ABB RAPID module: Module1.mod

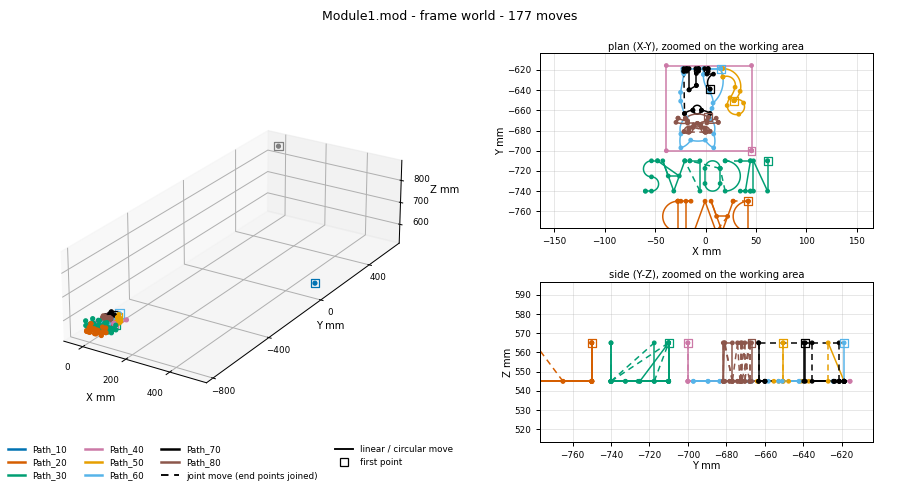
[picture p0: tool path of Module1.mod in frame world, 177 of 177 moves have a stored position in this frame; points joined in program order, loops and branches not executed]
MODULE Module1
    CONST robtarget Target_home:=[[-424.990093119,-612,35.499184826],[0,0.996194698,0,0.087155743],[0,0,0,0],[9E+09,9E+09,9E+09,9E+09,9E+09,9E+09]];
    CONST robtarget D1A:=[[68.121,138,20],[0,-0.707106781,0.707106781,0],[0,0,0,0],[9E+09,9E+09,9E+09,9E+09,9E+09,9E+09]];
    CONST robtarget D11:=[[68.121,138,0],[0,-0.707106781,0.707106781,0],[0,0,0,0],[9E+09,9E+09,9E+09,9E+09,9E+09,9E+09]];
    CONST robtarget D12:=[[68.121,168,0],[0,-0.707106781,0.707106781,0],[0,0,0,0],[9E+09,9E+09,9E+09,9E+09,9E+09,9E+09]];
    CONST robtarget D13:=[[83.121,153,0],[0,-0.707106781,0.707106781,0],[0,0,0,0],[9E+09,9E+09,9E+09,9E+09,9E+09,9E+09]];
    CONST robtarget A1A:=[[83.121,138,20],[0,-0.707106781,0.707106781,0],[0,0,0,0],[9E+09,9E+09,9E+09,9E+09,9E+09,9E+09]];
    CONST robtarget A11:=[[83.121,138,0],[0,-0.707106781,0.707106781,0],[0,0,0,0],[9E+09,9E+09,9E+09,9E+09,9E+09,9E+09]];
    CONST robtarget A12:=[[94.04,168,0],[0,-0.707106781,0.707106781,0],[0,0,0,0],[9E+09,9E+09,9E+09,9E+09,9E+09,9E+09]];
    CONST robtarget A13:=[[104.96,138,0],[0,-0.707106781,0.707106781,0],[0,0,0,0],[9E+09,9E+09,9E+09,9E+09,9E+09,9E+09]];
    CONST robtarget A14:=[[99.5,153,0],[0,-0.707106781,0.707106781,0],[0,0,0,0],[9E+09,9E+09,9E+09,9E+09,9E+09,9E+09]];
    CONST robtarget A15:=[[88.581,153,0],[0,-0.707106781,0.707106781,0],[0,0,0,0],[9E+09,9E+09,9E+09,9E+09,9E+09,9E+09]];
    CONST robtarget VA:=[[100.04,168,20],[0,-0.707106781,0.707106781,0],[0,0,0,0],[9E+09,9E+09,9E+09,9E+09,9E+09,9E+09]];
    CONST robtarget V1:=[[100.04,168,0],[0,-0.707106781,0.707106781,0],[0,0,0,0],[9E+09,9E+09,9E+09,9E+09,9E+09,9E+09]];
    CONST robtarget V2:=[[110.96,138,0],[0,-0.707106781,0.707106781,0],[0,0,0,0],[9E+09,9E+09,9E+09,9E+09,9E+09,9E+09]];
    CONST robtarget V3:=[[121.879,168,0],[0,-0.707106781,0.707106781,0],[0,0,0,0],[9E+09,9E+09,9E+09,9E+09,9E+09,9E+09]];
    CONST robtarget I1A:=[[124.879,168,20],[0,-0.707106781,0.707106781,0],[0,0,0,0],[9E+09,9E+09,9E+09,9E+09,9E+09,9E+09]];
    CONST robtarget I11:=[[124.879,168,0],[0,-0.707106781,0.707106781,0],[0,0,0,0],[9E+09,9E+09,9E+09,9E+09,9E+09,9E+09]];
    CONST robtarget I12:=[[134.879,168,0],[0,-0.707106781,0.707106781,0],[0,0,0,0],[9E+09,9E+09,9E+09,9E+09,9E+09,9E+09]];
    CONST robtarget I13:=[[129.879,168,0],[0,-0.707106781,0.707106781,0],[0,0,0,0],[9E+09,9E+09,9E+09,9E+09,9E+09,9E+09]];
    CONST robtarget I14:=[[129.879,138,0],[0,-0.707106781,0.707106781,0],[0,0,0,0],[9E+09,9E+09,9E+09,9E+09,9E+09,9E+09]];
    CONST robtarget I15:=[[124.879,138,0],[0,-0.707106781,0.707106781,0],[0,0,0,0],[9E+09,9E+09,9E+09,9E+09,9E+09,9E+09]];
    CONST robtarget I16:=[[134.879,138,0],[0,-0.707106781,0.707106781,0],[0,0,0,0],[9E+09,9E+09,9E+09,9E+09,9E+09,9E+09]];
    CONST robtarget D2A:=[[137.879,138,20],[0,-0.707106781,0.707106781,0],[0,0,0,0],[9E+09,9E+09,9E+09,9E+09,9E+09,9E+09]];
    CONST robtarget D21:=[[137.879,138,0],[0,-0.707106781,0.707106781,0],[0,0,0,0],[9E+09,9E+09,9E+09,9E+09,9E+09,9E+09]];
    CONST robtarget D22:=[[137.879,168,0],[0,-0.707106781,0.707106781,0],[0,0,0,0],[9E+09,9E+09,9E+09,9E+09,9E+09,9E+09]];
    CONST robtarget D23:=[[152.879,153,0],[0,-0.707106781,0.707106781,0],[0,0,0,0],[9E+09,9E+09,9E+09,9E+09,9E+09,9E+09]];
    PERS tooldata PM:=[TRUE,[[71.138,0,74.787],[0.819152044,0,0.573576436,0]],[1,[0,0,1],[1,0,0,0],0,0,0]];
    TASK PERS wobjdata Pastel:=[FALSE,TRUE,"",[[0,0,0],[1,0,0,0]],[[110.5,-612,545],[0,0,0,1]]];
    CONST robtarget SA:=[[158.029,98,20],[0,-0.707106781,0.707106781,0],[0,0,0,0],[9E+09,9E+09,9E+09,9E+09,9E+09,9E+09]];
    CONST robtarget CA:=[[91.029,98,20],[0,-0.707106781,0.707106781,0],[0,0,0,0],[9E+09,9E+09,9E+09,9E+09,9E+09,9E+09]];
    CONST robtarget C1:=[[91.029,98,0],[0,-0.707106781,0.707106781,0],[0,0,0,0],[9E+09,9E+09,9E+09,9E+09,9E+09,9E+09]];
    CONST robtarget C2:=[[76.029,113,0],[0,-0.707106781,0.707106781,0],[0,0,0,0],[9E+09,9E+09,9E+09,9E+09,9E+09,9E+09]];
    CONST robtarget C3:=[[91.029,128,0],[0,-0.707106781,0.707106781,0],[0,0,0,0],[9E+09,9E+09,9E+09,9E+09,9E+09,9E+09]];
    CONST robtarget OA:=[[96.029,105.5,20],[0,-0.707106781,0.707106781,0],[0,0,0,0],[9E+09,9E+09,9E+09,9E+09,9E+09,9E+09]];
    CONST robtarget O1:=[[96.029,105.5,0],[0,-0.707106781,0.707106781,0],[0,0,0,0],[9E+09,9E+09,9E+09,9E+09,9E+09,9E+09]];
    CONST robtarget O2:=[[96.029,120.5,0],[0,-0.707106781,0.707106781,0],[0,0,0,0],[9E+09,9E+09,9E+09,9E+09,9E+09,9E+09]];
    CONST robtarget O3:=[[103.529,128,0],[0,-0.707106781,0.707106781,0],[0,0,0,0],[9E+09,9E+09,9E+09,9E+09,9E+09,9E+09]];
    CONST robtarget O4:=[[111.029,120.5,0],[0,-0.707106781,0.707106781,0],[0,0,0,0],[9E+09,9E+09,9E+09,9E+09,9E+09,9E+09]];
    CONST robtarget O5:=[[111.029,105.5,0],[0,-0.707106781,0.707106781,0],[0,0,0,0],[9E+09,9E+09,9E+09,9E+09,9E+09,9E+09]];
    CONST robtarget O6:=[[103.529,98,0],[0,-0.707106781,0.707106781,0],[0,0,0,0],[9E+09,9E+09,9E+09,9E+09,9E+09,9E+09]];
    CONST robtarget LA:=[[126.029,98,20],[0,-0.707106781,0.707106781,0],[0,0,0,0],[9E+09,9E+09,9E+09,9E+09,9E+09,9E+09]];
    CONST robtarget L1:=[[126.029,98,0],[0,-0.707106781,0.707106781,0],[0,0,0,0],[9E+09,9E+09,9E+09,9E+09,9E+09,9E+09]];
    CONST robtarget L2:=[[116.029,98,0],[0,-0.707106781,0.707106781,0],[0,0,0,0],[9E+09,9E+09,9E+09,9E+09,9E+09,9E+09]];
    CONST robtarget L3:=[[116.029,128,0],[0,-0.707106781,0.707106781,0],[0,0,0,0],[9E+09,9E+09,9E+09,9E+09,9E+09,9E+09]];
    CONST robtarget A2A:=[[131.029,98,20],[0,-0.707106781,0.707106781,0],[0,0,0,0],[9E+09,9E+09,9E+09,9E+09,9E+09,9E+09]];
    CONST robtarget A21:=[[131.029,98,0],[0,-0.707106781,0.707106781,0],[0,0,0,0],[9E+09,9E+09,9E+09,9E+09,9E+09,9E+09]];
    CONST robtarget A22:=[[141.948,128,0],[0,-0.707106781,0.707106781,0],[0,0,0,0],[9E+09,9E+09,9E+09,9E+09,9E+09,9E+09]];
    CONST robtarget A23:=[[152.867,98,0],[0,-0.707106781,0.707106781,0],[0,0,0,0],[9E+09,9E+09,9E+09,9E+09,9E+09,9E+09]];
    CONST robtarget A24:=[[147.408,113,0],[0,-0.707106781,0.707106781,0],[0,0,0,0],[9E+09,9E+09,9E+09,9E+09,9E+09,9E+09]];
    CONST robtarget A25:=[[136.489,113,0],[0,-0.707106781,0.707106781,0],[0,0,0,0],[9E+09,9E+09,9E+09,9E+09,9E+09,9E+09]];
    CONST robtarget S1:=[[158.029,98,0],[0,-0.707106781,0.707106781,0],[0,0,0,0],[9E+09,9E+09,9E+09,9E+09,9E+09,9E+09]];
    CONST robtarget S2:=[[164.029,98,0],[0,-0.707106781,0.707106781,0],[0,0,0,0],[9E+09,9E+09,9E+09,9E+09,9E+09,9E+09]];
    CONST robtarget S3:=[[171.971,105.942,0],[0,-0.707106781,0.707106781,0],[0,0,0,0],[9E+09,9E+09,9E+09,9E+09,9E+09,9E+09]];
    CONST robtarget S4:=[[164.029,113.883,0],[0,-0.707106781,0.707106781,0],[0,0,0,0],[9E+09,9E+09,9E+09,9E+09,9E+09,9E+09]];
    CONST robtarget S5:=[[156.971,120.942,0],[0,-0.707106781,0.707106781,0],[0,0,0,0],[9E+09,9E+09,9E+09,9E+09,9E+09,9E+09]];
    CONST robtarget S6:=[[164.029,128,0],[0,-0.707106781,0.707106781,0],[0,0,0,0],[9E+09,9E+09,9E+09,9E+09,9E+09,9E+09]];
    CONST robtarget S7:=[[170.029,128,0],[0,-0.707106781,0.707106781,0],[0,0,0,0],[9E+09,9E+09,9E+09,9E+09,9E+09,9E+09]];
    CONST robtarget SF:=[[170.029,128,20],[0,-0.707106781,0.707106781,0],[0,0,0,0],[9E+09,9E+09,9E+09,9E+09,9E+09,9E+09]];
    CONST robtarget NA:=[[49.029,98,20],[0,-0.707106781,0.707106781,0],[0,0,0,0],[9E+09,9E+09,9E+09,9E+09,9E+09,9E+09]];
    CONST robtarget N4:=[[63.029,128,0],[0,-0.707106781,0.707106781,0],[0,0,0,0],[9E+09,9E+09,9E+09,9E+09,9E+09,9E+09]];
    CONST robtarget N3:=[[63.029,98,0],[0,-0.707106781,0.707106781,0],[0,0,0,0],[9E+09,9E+09,9E+09,9E+09,9E+09,9E+09]];
    CONST robtarget N2:=[[49.029,128,0],[0,-0.707106781,0.707106781,0],[0,0,0,0],[9E+09,9E+09,9E+09,9E+09,9E+09,9E+09]];
    CONST robtarget N1:=[[49.029,98,0],[0,-0.707106781,0.707106781,0],[0,0,0,0],[9E+09,9E+09,9E+09,9E+09,9E+09,9E+09]];
    CONST robtarget I26:=[[76.029,98,0],[0,-0.707106781,0.707106781,0],[0,0,0,0],[9E+09,9E+09,9E+09,9E+09,9E+09,9E+09]];
    CONST robtarget I25:=[[66.029,98,0],[0,-0.707106781,0.707106781,0],[0,0,0,0],[9E+09,9E+09,9E+09,9E+09,9E+09,9E+09]];
    CONST robtarget I24:=[[71.029,98,0],[0,-0.707106781,0.707106781,0],[0,0,0,0],[9E+09,9E+09,9E+09,9E+09,9E+09,9E+09]];
    CONST robtarget I23:=[[71.029,128,0],[0,-0.707106781,0.707106781,0],[0,0,0,0],[9E+09,9E+09,9E+09,9E+09,9E+09,9E+09]];
    CONST robtarget I22:=[[76.029,128,0],[0,-0.707106781,0.707106781,0],[0,0,0,0],[9E+09,9E+09,9E+09,9E+09,9E+09,9E+09]];
    CONST robtarget I21:=[[66.029,128,0],[0,-0.707106781,0.707106781,0],[0,0,0,0],[9E+09,9E+09,9E+09,9E+09,9E+09,9E+09]];
    CONST robtarget I2A:=[[66.029,128,20],[0,-0.707106781,0.707106781,0],[0,0,0,0],[9E+09,9E+09,9E+09,9E+09,9E+09,9E+09]];
    CONST robtarget CUAA:=[[64.919,88,20],[0,-0.707106781,0.707106781,0],[0,0,0,0],[9E+09,9E+09,9E+09,9E+09,9E+09,9E+09]];
    CONST robtarget E1:=[[64.919,88,0],[0,-0.707106781,0.707106781,0],[0,0,0,0],[9E+09,9E+09,9E+09,9E+09,9E+09,9E+09]];
    CONST robtarget E2:=[[149.319,88,0],[0,-0.707106781,0.707106781,0],[0,0,0,0],[9E+09,9E+09,9E+09,9E+09,9E+09,9E+09]];
    CONST robtarget E3:=[[149.319,3.6,0],[0,-0.707106781,0.707106781,0],[0,0,0,0],[9E+09,9E+09,9E+09,9E+09,9E+09,9E+09]];
    CONST robtarget E4:=[[64.919,3.6,0],[0,-0.707106781,0.707106781,0],[0,0,0,0],[9E+09,9E+09,9E+09,9E+09,9E+09,9E+09]];
    CONST robtarget P11:=[[82.21,38.425,20],[0,-0.707106781,0.707106781,0],[0,0,0,0],[9E+09,9E+09,9E+09,9E+09,9E+09,9E+09]];
    CONST robtarget P12:=[[82.21,38.425,0],[0,-0.707106781,0.707106781,0],[0,0,0,0],[9E+09,9E+09,9E+09,9E+09,9E+09,9E+09]];
    CONST robtarget P13:=[[76.99,37.487,0],[0,-0.707106781,0.707106781,0],[0,0,0,0],[9E+09,9E+09,9E+09,9E+09,9E+09,9E+09]];
    CONST robtarget P14:=[[72.798,40.737,0],[0,-0.707106781,0.707106781,0],[0,0,0,0],[9E+09,9E+09,9E+09,9E+09,9E+09,9E+09]];
    CONST robtarget P15:=[[72.498,47.446,0],[0,-0.707106781,0.707106781,0],[0,0,0,0],[9E+09,9E+09,9E+09,9E+09,9E+09,9E+09]];
    CONST robtarget P16:=[[77.549,51.872,0],[0,-0.707106781,0.707106781,0],[0,0,0,0],[9E+09,9E+09,9E+09,9E+09,9E+09,9E+09]];
    CONST robtarget P17:=[[85.419,50.387,0],[0,-0.707106781,0.707106781,0],[0,0,0,0],[9E+09,9E+09,9E+09,9E+09,9E+09,9E+09]];
    CONST robtarget P18:=[[89.032,43.239,0],[0,-0.707106781,0.707106781,0],[0,0,0,0],[9E+09,9E+09,9E+09,9E+09,9E+09,9E+09]];
    CONST robtarget P19:=[[88.217,39.173,0],[0,-0.707106781,0.707106781,0],[0,0,0,0],[9E+09,9E+09,9E+09,9E+09,9E+09,9E+09]];
    CONST robtarget P110:=[[86.183,35.559,0],[0,-0.707106781,0.707106781,0],[0,0,0,0],[9E+09,9E+09,9E+09,9E+09,9E+09,9E+09]];
    CONST robtarget P111:=[[83.19,30.571,0],[0,-0.707106781,0.707106781,0],[0,0,0,0],[9E+09,9E+09,9E+09,9E+09,9E+09,9E+09]];
    CONST robtarget P112:=[[81.2,25.106,0],[0,-0.707106781,0.707106781,0],[0,0,0,0],[9E+09,9E+09,9E+09,9E+09,9E+09,9E+09]];
    CONST robtarget P113:=[[84.037,16.23,0],[0,-0.707106781,0.707106781,0],[0,0,0,0],[9E+09,9E+09,9E+09,9E+09,9E+09,9E+09]];
    CONST robtarget P114:=[[93.269,14.968,0],[0,-0.707106781,0.707106781,0],[0,0,0,0],[9E+09,9E+09,9E+09,9E+09,9E+09,9E+09]];
    CONST robtarget P115:=[[93.269,14.968,20],[0,-0.707106781,0.707106781,0],[0,0,0,0],[9E+09,9E+09,9E+09,9E+09,9E+09,9E+09]];
    CONST robtarget P116:=[[95.609,6.67,0],[0,-0.707106781,0.707106781,0],[0,0,0,0],[9E+09,9E+09,9E+09,9E+09,9E+09,9E+09]];
    CONST robtarget P117:=[[93.269,6.67,0],[0,-0.707106781,0.707106781,0],[0,0,0,0],[9E+09,9E+09,9E+09,9E+09,9E+09,9E+09]];
    CONST robtarget P118:=[[79.171,13.675,0],[0,-0.707106781,0.707106781,0],[0,0,0,0],[9E+09,9E+09,9E+09,9E+09,9E+09,9E+09]];
    CONST robtarget P119:=[[76.238,29.142,0],[0,-0.707106781,0.707106781,0],[0,0,0,0],[9E+09,9E+09,9E+09,9E+09,9E+09,9E+09]];
    CONST robtarget P120:=[[78.528,34.232,0],[0,-0.707106781,0.707106781,0],[0,0,0,0],[9E+09,9E+09,9E+09,9E+09,9E+09,9E+09]];
    CONST robtarget P232:=[[103.027,40.737,0],[0,-0.707106781,0.707106781,0],[0,0,0,0],[9E+09,9E+09,9E+09,9E+09,9E+09,9E+09]];
    CONST robtarget P210:=[[135.23,62.86,0],[0,-0.707106781,0.707106781,0],[0,0,0,0],[9E+09,9E+09,9E+09,9E+09,9E+09,9E+09]];
    CONST robtarget P211:=[[134.911,71.377,0],[0,-0.707106781,0.707106781,0],[0,0,0,0],[9E+09,9E+09,9E+09,9E+09,9E+09,9E+09]];
    CONST robtarget P212:=[[135.861,78.258,0],[0,-0.707106781,0.707106781,0],[0,0,0,0],[9E+09,9E+09,9E+09,9E+09,9E+09,9E+09]];
    CONST robtarget P213:=[[134.911,85.138,0],[0,-0.707106781,0.707106781,0],[0,0,0,0],[9E+09,9E+09,9E+09,9E+09,9E+09,9E+09]];
    CONST robtarget P214:=[[129.352,82.199,0],[0,-0.707106781,0.707106781,0],[0,0,0,0],[9E+09,9E+09,9E+09,9E+09,9E+09,9E+09]];
    CONST robtarget P215:=[[125.181,77.493,0],[0,-0.707106781,0.707106781,0],[0,0,0,0],[9E+09,9E+09,9E+09,9E+09,9E+09,9E+09]];
    CONST robtarget P216:=[[117.953,78.45,0],[0,-0.707106781,0.707106781,0],[0,0,0,0],[9E+09,9E+09,9E+09,9E+09,9E+09,9E+09]];
    CONST robtarget P217:=[[110.724,77.493,0],[0,-0.707106781,0.707106781,0],[0,0,0,0],[9E+09,9E+09,9E+09,9E+09,9E+09,9E+09]];
    CONST robtarget P218:=[[107.111,81.908,0],[0,-0.707106781,0.707106781,0],[0,0,0,0],[9E+09,9E+09,9E+09,9E+09,9E+09,9E+09]];
    CONST robtarget P219:=[[102.4,85.125,0],[0,-0.707106781,0.707106781,0],[0,0,0,0],[9E+09,9E+09,9E+09,9E+09,9E+09,9E+09]];
    CONST robtarget P220:=[[101.194,78.244,0],[0,-0.707106781,0.707106781,0],[0,0,0,0],[9E+09,9E+09,9E+09,9E+09,9E+09,9E+09]];
    CONST robtarget P221:=[[102.4,71.363,0],[0,-0.707106781,0.707106781,0],[0,0,0,0],[9E+09,9E+09,9E+09,9E+09,9E+09,9E+09]];
    CONST robtarget P222:=[[101.604,63.136,0],[0,-0.707106781,0.707106781,0],[0,0,0,0],[9E+09,9E+09,9E+09,9E+09,9E+09,9E+09]];
    CONST robtarget P223:=[[105.943,56.102,0],[0,-0.707106781,0.707106781,0],[0,0,0,0],[9E+09,9E+09,9E+09,9E+09,9E+09,9E+09]];
    CONST robtarget P224:=[[107.614,54.857,0],[0,-0.707106781,0.707106781,0],[0,0,0,0],[9E+09,9E+09,9E+09,9E+09,9E+09,9E+09]];
    CONST robtarget P225:=[[104.069,46.093,0],[0,-0.707106781,0.707106781,0],[0,0,0,0],[9E+09,9E+09,9E+09,9E+09,9E+09,9E+09]];
    CONST robtarget P226:=[[103.223,37.713,0],[0,-0.707106781,0.707106781,0],[0,0,0,0],[9E+09,9E+09,9E+09,9E+09,9E+09,9E+09]];
    CONST robtarget P227:=[[106.607,30,0],[0,-0.707106781,0.707106781,0],[0,0,0,0],[9E+09,9E+09,9E+09,9E+09,9E+09,9E+09]];
    CONST robtarget P228:=[[111.198,21.776,0],[0,-0.707106781,0.707106781,0],[0,0,0,0],[9E+09,9E+09,9E+09,9E+09,9E+09,9E+09]];
    CONST robtarget P229:=[[112.662,12.472,0],[0,-0.707106781,0.707106781,0],[0,0,0,0],[9E+09,9E+09,9E+09,9E+09,9E+09,9E+09]];
    CONST robtarget P230:=[[112.476,6.67,0],[0,-0.707106781,0.707106781,0],[0,0,0,0],[9E+09,9E+09,9E+09,9E+09,9E+09,9E+09]];
    CONST robtarget P231:=[[93.703,24.926,0],[0,-0.707106781,0.707106781,0],[0,0,0,0],[9E+09,9E+09,9E+09,9E+09,9E+09,9E+09]];
    CONST robtarget P29:=[[129.718,55.201,0],[0,-0.707106781,0.707106781,0],[0,0,0,0],[9E+09,9E+09,9E+09,9E+09,9E+09,9E+09]];
    CONST robtarget P28:=[[132.81,47.291,0],[0,-0.707106781,0.707106781,0],[0,0,0,0],[9E+09,9E+09,9E+09,9E+09,9E+09,9E+09]];
    CONST robtarget P27:=[[135.088,38.885,0],[0,-0.707106781,0.707106781,0],[0,0,0,0],[9E+09,9E+09,9E+09,9E+09,9E+09,9E+09]];
    CONST robtarget P26:=[[135.236,30.178,0],[0,-0.707106781,0.707106781,0],[0,0,0,0],[9E+09,9E+09,9E+09,9E+09,9E+09,9E+09]];
    CONST robtarget P25:=[[131.968,12.02,0],[0,-0.707106781,0.707106781,0],[0,0,0,0],[9E+09,9E+09,9E+09,9E+09,9E+09,9E+09]];
    CONST robtarget P24:=[[134.388,9.719,0],[0,-0.707106781,0.707106781,0],[0,0,0,0],[9E+09,9E+09,9E+09,9E+09,9E+09,9E+09]];
    CONST robtarget P23:=[[133.026,6.67,0],[0,-0.707106781,0.707106781,0],[0,0,0,0],[9E+09,9E+09,9E+09,9E+09,9E+09,9E+09]];
    CONST robtarget P22:=[[95.609,6.67,0],[0,-0.707106781,0.707106781,0],[0,0,0,0],[9E+09,9E+09,9E+09,9E+09,9E+09,9E+09]];
    CONST robtarget P21:=[[95.609,6.67,20],[0,-0.707106781,0.707106781,0],[0,0,0,0],[9E+09,9E+09,9E+09,9E+09,9E+09,9E+09]];
    CONST robtarget P31:=[[106.008,26.905,20],[0,-0.707106781,0.707106781,0],[0,0,0,0],[9E+09,9E+09,9E+09,9E+09,9E+09,9E+09]];
    CONST robtarget P32:=[[106.008,26.905,0],[0,-0.707106781,0.707106781,0],[0,0,0,0],[9E+09,9E+09,9E+09,9E+09,9E+09,9E+09]];
    CONST robtarget P33:=[[108.265,18.63,0],[0,-0.707106781,0.707106781,0],[0,0,0,0],[9E+09,9E+09,9E+09,9E+09,9E+09,9E+09]];
    CONST robtarget P34:=[[102.665,12.134,0],[0,-0.707106781,0.707106781,0],[0,0,0,0],[9E+09,9E+09,9E+09,9E+09,9E+09,9E+09]];
    CONST robtarget P35:=[[109.043,12.02,0],[0,-0.707106781,0.707106781,0],[0,0,0,0],[9E+09,9E+09,9E+09,9E+09,9E+09,9E+09]];
    CONST robtarget P36:=[[111.486,9.9,0],[0,-0.707106781,0.707106781,0],[0,0,0,0],[9E+09,9E+09,9E+09,9E+09,9E+09,9E+09]];
    CONST robtarget P37:=[[111.341,6.67,0],[0,-0.707106781,0.707106781,0],[0,0,0,0],[9E+09,9E+09,9E+09,9E+09,9E+09,9E+09]];
    CONST robtarget P38:=[[107.849,6.67,0],[0,-0.707106781,0.707106781,0],[0,0,0,0],[9E+09,9E+09,9E+09,9E+09,9E+09,9E+09]];
    CONST robtarget P39:=[[107.849,9.239,0],[0,-0.707106781,0.707106781,0],[0,0,0,0],[9E+09,9E+09,9E+09,9E+09,9E+09,9E+09]];
    CONST robtarget P310:=[[117.381,6.67,0],[0,-0.707106781,0.707106781,0],[0,0,0,0],[9E+09,9E+09,9E+09,9E+09,9E+09,9E+09]];
    CONST robtarget P311:=[[117.381,9.136,0],[0,-0.707106781,0.707106781,0],[0,0,0,0],[9E+09,9E+09,9E+09,9E+09,9E+09,9E+09]];
    CONST robtarget P312:=[[120.124,6.67,0],[0,-0.707106781,0.707106781,0],[0,0,0,0],[9E+09,9E+09,9E+09,9E+09,9E+09,9E+09]];
    CONST robtarget P313:=[[121.413,9.237,0],[0,-0.707106781,0.707106781,0],[0,0,0,0],[9E+09,9E+09,9E+09,9E+09,9E+09,9E+09]];
    CONST robtarget P314:=[[119.569,11.44,0],[0,-0.707106781,0.707106781,0],[0,0,0,0],[9E+09,9E+09,9E+09,9E+09,9E+09,9E+09]];
    CONST robtarget P315:=[[119.569,23.339,0],[0,-0.707106781,0.707106781,0],[0,0,0,0],[9E+09,9E+09,9E+09,9E+09,9E+09,9E+09]];
    CONST robtarget P316:=[[119.569,23.339,20],[0,-0.707106781,0.707106781,0],[0,0,0,0],[9E+09,9E+09,9E+09,9E+09,9E+09,9E+09]];
    CONST robtarget P317:=[[126.788,27.654,20],[0,-0.707106781,0.707106781,0],[0,0,0,0],[9E+09,9E+09,9E+09,9E+09,9E+09,9E+09]];
    CONST robtarget P318:=[[126.788,27.654,0],[0,-0.707106781,0.707106781,0],[0,0,0,0],[9E+09,9E+09,9E+09,9E+09,9E+09,9E+09]];
    CONST robtarget P319:=[[126.788,6.67,0],[0,-0.707106781,0.707106781,0],[0,0,0,0],[9E+09,9E+09,9E+09,9E+09,9E+09,9E+09]];
    CONST robtarget P320:=[[129.217,6.67,0],[0,-0.707106781,0.707106781,0],[0,0,0,0],[9E+09,9E+09,9E+09,9E+09,9E+09,9E+09]];
    CONST robtarget P321:=[[129.217,9.26,0],[0,-0.707106781,0.707106781,0],[0,0,0,0],[9E+09,9E+09,9E+09,9E+09,9E+09,9E+09]];
    CONST robtarget P322:=[[131.968,6.67,0],[0,-0.707106781,0.707106781,0],[0,0,0,0],[9E+09,9E+09,9E+09,9E+09,9E+09,9E+09]];
    CONST robtarget P323:=[[131.968,9.288,0],[0,-0.707106781,0.707106781,0],[0,0,0,0],[9E+09,9E+09,9E+09,9E+09,9E+09,9E+09]];
    CONST robtarget P324:=[[131.968,9.288,20],[0,-0.707106781,0.707106781,0],[0,0,0,0],[9E+09,9E+09,9E+09,9E+09,9E+09,9E+09]];
    CONST robtarget P325:=[[131.291,51.178,20],[0,-0.707106781,0.707106781,0],[0,0,0,0],[9E+09,9E+09,9E+09,9E+09,9E+09,9E+09]];
    CONST robtarget P326:=[[131.291,51.178,0],[0,-0.707106781,0.707106781,0],[0,0,0,0],[9E+09,9E+09,9E+09,9E+09,9E+09,9E+09]];
    CONST robtarget P327:=[[127.419,48.872,0],[0,-0.707106781,0.707106781,0],[0,0,0,0],[9E+09,9E+09,9E+09,9E+09,9E+09,9E+09]];
    CONST robtarget P328:=[[123.025,47.87,0],[0,-0.707106781,0.707106781,0],[0,0,0,0],[9E+09,9E+09,9E+09,9E+09,9E+09,9E+09]];
    CONST robtarget P329:=[[118.76,42.987,0],[0,-0.707106781,0.707106781,0],[0,0,0,0],[9E+09,9E+09,9E+09,9E+09,9E+09,9E+09]];
    CONST robtarget P330:=[[114.503,47.934,0],[0,-0.707106781,0.707106781,0],[0,0,0,0],[9E+09,9E+09,9E+09,9E+09,9E+09,9E+09]];
    CONST robtarget P331:=[[118.76,51.596,0],[0,-0.707106781,0.707106781,0],[0,0,0,0],[9E+09,9E+09,9E+09,9E+09,9E+09,9E+09]];
    CONST robtarget P332:=[[106.12,51.162,20],[0,-0.707106781,0.707106781,0],[0,0,0,0],[9E+09,9E+09,9E+09,9E+09,9E+09,9E+09]];
    CONST robtarget P333:=[[106.12,51.162,0],[0,-0.707106781,0.707106781,0],[0,0,0,0],[9E+09,9E+09,9E+09,9E+09,9E+09,9E+09]];
    CONST robtarget P334:=[[110.069,48.918,0],[0,-0.707106781,0.707106781,0],[-1,-1,0,0],[9E+09,9E+09,9E+09,9E+09,9E+09,9E+09]];
    CONST robtarget Target_390:=[[106.06,68.753,20],[0,-0.707106781,0.707106781,0],[0,0,0,0],[9E+09,9E+09,9E+09,9E+09,9E+09,9E+09]];
    CONST robtarget Target_10:=[[107.614,54.857,20],[0,-0.707106781,0.707106781,0],[0,0,0,0],[9E+09,9E+09,9E+09,9E+09,9E+09,9E+09]];
    CONST robtarget Target_20:=[[107.614,54.857,0],[0,-0.707106781,0.707106781,0],[0,0,0,0],[9E+09,9E+09,9E+09,9E+09,9E+09,9E+09]];
    CONST robtarget Target_30:=[[118.158,51.596,0],[0,-0.707106781,0.707106781,0],[0,0,0,0],[9E+09,9E+09,9E+09,9E+09,9E+09,9E+09]];
    CONST robtarget Target_40:=[[130.488,55.777,0],[0,-0.707106781,0.707106781,0],[0,0,0,0],[9E+09,9E+09,9E+09,9E+09,9E+09,9E+09]];
    CONST robtarget Target_50:=[[130.488,55.777,20],[0,-0.707106781,0.707106781,0],[0,0,0,0],[9E+09,9E+09,9E+09,9E+09,9E+09,9E+09]];
    CONST robtarget Target_60:=[[128.271,58.346,0],[0,-0.707106781,0.707106781,0],[0,0,0,0],[9E+09,9E+09,9E+09,9E+09,9E+09,9E+09]];
    CONST robtarget Target_70:=[[133.152,57.611,0],[0,-0.707106781,0.707106781,0],[0,0,0,0],[9E+09,9E+09,9E+09,9E+09,9E+09,9E+09]];
    CONST robtarget Target_80:=[[137.735,55.777,0],[0,-0.707106781,0.707106781,0],[0,0,0,0],[9E+09,9E+09,9E+09,9E+09,9E+09,9E+09]];
    CONST robtarget Target_90:=[[137.735,55.777,20],[0,-0.707106781,0.707106781,0],[0,0,0,0],[9E+09,9E+09,9E+09,9E+09,9E+09,9E+09]];
    CONST robtarget Target_100:=[[139.742,59.868,0],[0,-0.707106781,0.707106781,0],[0,0,0,0],[9E+09,9E+09,9E+09,9E+09,9E+09,9E+09]];
    CONST robtarget Target_110:=[[134.046,60.945,0],[0,-0.707106781,0.707106781,0],[0,0,0,0],[9E+09,9E+09,9E+09,9E+09,9E+09,9E+09]];
    CONST robtarget Target_120:=[[128.271,60.458,0],[0,-0.707106781,0.707106781,0],[0,0,0,0],[9E+09,9E+09,9E+09,9E+09,9E+09,9E+09]];
    CONST robtarget Target_130:=[[128.271,60.458,20],[0,-0.707106781,0.707106781,0],[0,0,0,0],[9E+09,9E+09,9E+09,9E+09,9E+09,9E+09]];
    CONST robtarget Target_140:=[[109.172,60.458,0],[0,-0.707106781,0.707106781,0],[0,0,0,0],[9E+09,9E+09,9E+09,9E+09,9E+09,9E+09]];
    CONST robtarget Target_150:=[[103.474,60.737,0],[0,-0.707106781,0.707106781,0],[0,0,0,0],[9E+09,9E+09,9E+09,9E+09,9E+09,9E+09]];
    CONST robtarget Target_160:=[[97.835,59.868,0],[0,-0.707106781,0.707106781,0],[0,0,0,0],[9E+09,9E+09,9E+09,9E+09,9E+09,9E+09]];
    CONST robtarget Target_170:=[[97.835,59.868,20],[0,-0.707106781,0.707106781,0],[0,0,0,0],[9E+09,9E+09,9E+09,9E+09,9E+09,9E+09]];
    CONST robtarget Target_180:=[[99.9,55.777,0],[0,-0.707106781,0.707106781,0],[0,0,0,0],[9E+09,9E+09,9E+09,9E+09,9E+09,9E+09]];
    CONST robtarget Target_190:=[[104.361,57.694,0],[0,-0.707106781,0.707106781,0],[0,0,0,0],[9E+09,9E+09,9E+09,9E+09,9E+09,9E+09]];
    CONST robtarget Target_200:=[[109.172,58.346,0],[0,-0.707106781,0.707106781,0],[0,0,0,0],[9E+09,9E+09,9E+09,9E+09,9E+09,9E+09]];
    CONST robtarget Target_210:=[[109.172,58.346,20],[0,-0.707106781,0.707106781,0],[0,0,0,0],[9E+09,9E+09,9E+09,9E+09,9E+09,9E+09]];
    CONST robtarget Target_220:=[[118.604,60.887,0],[0,-0.707106781,0.707106781,0],[0,0,0,0],[9E+09,9E+09,9E+09,9E+09,9E+09,9E+09]];
    CONST robtarget Target_230:=[[121.915,62.126,0],[0,-0.707106781,0.707106781,0],[0,0,0,0],[9E+09,9E+09,9E+09,9E+09,9E+09,9E+09]];
    CONST robtarget Target_240:=[[118.609,64.422,0],[0,-0.707106781,0.707106781,0],[0,0,0,0],[9E+09,9E+09,9E+09,9E+09,9E+09,9E+09]];
    CONST robtarget Target_250:=[[115.296,62.135,0],[0,-0.707106781,0.707106781,0],[0,0,0,0],[9E+09,9E+09,9E+09,9E+09,9E+09,9E+09]];
    CONST robtarget Target_260:=[[115.296,62.135,20],[0,-0.707106781,0.707106781,0],[0,0,0,0],[9E+09,9E+09,9E+09,9E+09,9E+09,9E+09]];
    CONST robtarget Target_270:=[[114.503,64.832,0],[0,-0.707106781,0.707106781,0],[0,0,0,0],[9E+09,9E+09,9E+09,9E+09,9E+09,9E+09]];
    CONST robtarget Target_280:=[[109.172,64.403,0],[0,-0.707106781,0.707106781,0],[0,0,0,0],[9E+09,9E+09,9E+09,9E+09,9E+09,9E+09]];
    CONST robtarget Target_290:=[[111.574,70.748,0],[0,-0.707106781,0.707106781,0],[0,0,0,0],[9E+09,9E+09,9E+09,9E+09,9E+09,9E+09]];
    CONST robtarget Target_300:=[[125.272,70.252,0],[0,-0.707106781,0.707106781,0],[0,0,0,0],[9E+09,9E+09,9E+09,9E+09,9E+09,9E+09]];
    CONST robtarget Target_310:=[[127.174,63.734,0],[0,-0.707106781,0.707106781,0],[0,0,0,0],[9E+09,9E+09,9E+09,9E+09,9E+09,9E+09]];
    CONST robtarget Target_320:=[[110.609,66.183,0],[0,-0.707106781,0.707106781,0],[0,0,0,0],[9E+09,9E+09,9E+09,9E+09,9E+09,9E+09]];
    CONST robtarget Target_330:=[[127.028,66.212,0],[0,-0.707106781,0.707106781,0],[0,0,0,0],[9E+09,9E+09,9E+09,9E+09,9E+09,9E+09]];
    CONST robtarget Target_340:=[[106.06,68.753,0],[0,-0.707106781,0.707106781,0],[0,0,0,0],[9E+09,9E+09,9E+09,9E+09,9E+09,9E+09]];
    CONST robtarget Target_350:=[[123.025,64.832,0],[0,-0.707106781,0.707106781,0],[0,0,0,0],[9E+09,9E+09,9E+09,9E+09,9E+09,9E+09]];
    CONST robtarget Target_360:=[[131.721,69.031,0],[0,-0.707106781,0.707106781,0],[0,0,0,0],[9E+09,9E+09,9E+09,9E+09,9E+09,9E+09]];
    CONST robtarget Target_370:=[[123.025,64.832,20],[0,-0.707106781,0.707106781,0],[0,0,0,0],[9E+09,9E+09,9E+09,9E+09,9E+09,9E+09]];
    CONST robtarget Target_380:=[[131.721,69.031,20],[0,-0.707106781,0.707106781,0],[0,0,0,0],[9E+09,9E+09,9E+09,9E+09,9E+09,9E+09]];
    CONST robtarget Target_400:=[[110.609,69.551,20],[0,-0.707106781,0.707106781,0],[-2,0,-1,0],[9E+09,9E+09,9E+09,9E+09,9E+09,9E+09]];
    CONST robtarget Target_410:=[[110.609,69.551,0],[0,-0.707106781,0.707106781,0],[-2,0,-1,0],[9E+09,9E+09,9E+09,9E+09,9E+09,9E+09]];
    CONST robtarget Target_420:=[[127.028,69.522,0],[0,-0.707106781,0.707106781,0],[-2,0,-1,0],[9E+09,9E+09,9E+09,9E+09,9E+09,9E+09]];
    CONST robtarget Target_430:=[[127.028,69.522,20],[0,-0.707106781,0.707106781,0],[-2,0,-1,0],[9E+09,9E+09,9E+09,9E+09,9E+09,9E+09]];
    CONST robtarget Target_440:=[[112.284,68.043,0],[0,-0.707106781,0.707106781,0],[-2,0,-1,0],[9E+09,9E+09,9E+09,9E+09,9E+09,9E+09]];
    CONST robtarget Target_450:=[[110.609,66.183,0],[0,-0.707106781,0.707106781,0],[-2,0,-1,0],[9E+09,9E+09,9E+09,9E+09,9E+09,9E+09]];
    CONST robtarget Target_460:=[[108.935,67.691,0],[0,-0.707106781,0.707106781,0],[-1,-1,0,0],[9E+09,9E+09,9E+09,9E+09,9E+09,9E+09]];
    CONST robtarget Target_470:=[[128.679,67.98,0],[0,-0.707106781,0.707106781,0],[-2,0,-1,0],[9E+09,9E+09,9E+09,9E+09,9E+09,9E+09]];
    CONST robtarget Target_480:=[[127.028,66.212,0],[0,-0.707106781,0.707106781,0],[-2,0,-1,0],[9E+09,9E+09,9E+09,9E+09,9E+09,9E+09]];
    CONST robtarget Target_490:=[[125.376,67.952,0],[0,-0.707106781,0.707106781,0],[-2,0,-1,0],[9E+09,9E+09,9E+09,9E+09,9E+09,9E+09]];
    CONST robtarget Target_500:=[[107.716198612,-1209.812791745,313.527270399],[0.266060184,0.662603574,0.657812492,-0.239689817],[0,0,0,0],[9E+09,9E+09,9E+09,9E+09,9E+09,9E+09]];

    PROC main()
        RESET DO_01;
        RESET DO_02;
        WHILE TRUE DO
            IF DI_01 = 1 THEN
                SET DO_01;
                WaitTime 2;
                SET Conveyor_FWD;
                WaitTime 2;
                RESET Conveyor_FWD;
                Path_10;
                Path_10;
                Path_20;
                Path_30;
                Path_40;
                Path_50;
                Path_60;
                Path_70;
                Path_80;
                Path_10;
                WaitTime 2;
                SET Conveyor_FWD;
                WaitTime 2;
                RESET Conveyor_FWD;
                RESET DO_01;
            ELSEIF DI_02 = 1 THEN
                SET DO_02;
                Path_100;
                WHILE DI_03 = 0 DO
                ENDWHILE
                Path_10;
                RESET DO_02;
            ENDIF
        ENDWHILE
    ENDPROC

    PROC Path_10()

    MoveJ Target_home,v100,z10,PM\WObj:=Pastel;

    ENDPROC

    PROC Path_20()

        !!D!!
        MoveJ D1A,v100,z10,PM\WObj:=Pastel;
        MoveL D11,v100,z10,PM\WObj:=Pastel;
        MoveL D12,v100,z10,PM\WObj:=Pastel;
        MoveC D13,D11,v100,z10,PM\WObj:=Pastel;

        !!A!!
        MoveJ A1A,v100,z10,PM\WObj:=Pastel;
        MoveL A11,v100,z10,PM\WObj:=Pastel;
        MoveL A12,v100,z10,PM\WObj:=Pastel;
        MoveL A13,v100,z10,PM\WObj:=Pastel;
        MoveL A14,v100,z10,PM\WObj:=Pastel;
        MoveL A15,v100,z10,PM\WObj:=Pastel;

        !!V!!
        MoveJ VA,v100,z10,PM\WObj:=Pastel;
        MoveL V1,v100,z10,PM\WObj:=Pastel;
        MoveL V2,v100,z10,PM\WObj:=Pastel;
        MoveL V3,v100,z10,PM\WObj:=Pastel;

        !!I!!
        MoveJ I1A,v100,z10,PM\WObj:=Pastel;
        MoveL I11,v100,z10,PM\WObj:=Pastel;
        MoveL I12,v100,z10,PM\WObj:=Pastel;
        MoveL I13,v100,z10,PM\WObj:=Pastel;
        MoveL I14,v100,z10,PM\WObj:=Pastel;
        MoveL I15,v100,z10,PM\WObj:=Pastel;
        MoveL I16,v100,z10,PM\WObj:=Pastel;

        !!D!!
        MoveJ D2A,v100,z10,PM\WObj:=Pastel;
        MoveL D21,v100,z10,PM\WObj:=Pastel;
        MoveL D22,v100,z10,PM\WObj:=Pastel;
        MoveC D23,D21,v100,z10,PM\WObj:=Pastel;
        MoveJ D2A,v100,z10,PM\WObj:=Pastel;


    ENDPROC
    PROC Path_30()

        !!N!!
        MoveJ NA,v100,z10,PM\WObj:=Pastel;
        MoveL N1,v100,z10,PM\WObj:=Pastel;
        MoveL N2,v100,z10,PM\WObj:=Pastel;
        MoveL N3,v100,z10,PM\WObj:=Pastel;
        MoveL N4,v100,z10,PM\WObj:=Pastel;

        !!I!!
        MoveJ I2A,v100,z10,PM\WObj:=Pastel;
        MoveL I21,v100,z10,PM\WObj:=Pastel;
        MoveL I22,v100,z10,PM\WObj:=Pastel;
        MoveL I23,v100,z10,PM\WObj:=Pastel;
        MoveL I25,v100,z10,PM\WObj:=Pastel;
        MoveL I25,v100,z10,PM\WObj:=Pastel;
        MoveL I26,v100,z10,PM\WObj:=Pastel;

        !!C!!
        MoveJ CA,v100,z10,PM\WObj:=Pastel;
        MoveL C1,v100,z10,PM\WObj:=Pastel;
        MoveC C2,C3,v100,z10,PM\WObj:=Pastel;

        !!O!!
        MoveJ OA,v100,z10,PM\WObj:=Pastel;
        MoveL O1,v100,z10,PM\WObj:=Pastel;
        MoveL O2,v100,z10,PM\WObj:=Pastel;
        MoveC O3,O4,v100,z10,PM\WObj:=Pastel;
        MoveL O5,v100,z10,PM\WObj:=Pastel;
        MoveC O6,O1,v100,z10,PM\WObj:=Pastel;

        !!L!!
        MoveJ LA,v100,z10,PM\WObj:=Pastel;
        MoveL L1,v100,z10,PM\WObj:=Pastel;
        MoveL L2,v100,z10,PM\WObj:=Pastel;
        MoveL L3,v100,z10,PM\WObj:=Pastel;


        !!A!!
        MoveJ A2A,v100,z10,PM\WObj:=Pastel;
        MoveL A21,v100,z10,PM\WObj:=Pastel;
        MoveL A22,v100,z10,PM\WObj:=Pastel;
        MoveL A23,v100,z10,PM\WObj:=Pastel;
        MoveL A24,v100,z10,PM\WObj:=Pastel;
        MoveL A25,v100,z10,PM\WObj:=Pastel;

        !!S!!
        MoveL SA,v100,z10,PM\WObj:=Pastel;
        MoveL S1,v100,z10,PM\WObj:=Pastel;
        MoveL S2,v100,z10,PM\WObj:=Pastel;
        MoveC S3,S4,v100,z10,PM\WObj:=Pastel;
        MoveC S5,S6,v100,z10,PM\WObj:=Pastel;
        MoveL S7,v100,z10,PM\WObj:=Pastel;
        MoveL SF,v100,z10,PM\WObj:=Pastel;


    ENDPROC
    PROC Path_40()
        MoveJ CUAA,v100,z10,PM\WObj:=Pastel;
        MoveL E1,v100,z10,PM\WObj:=Pastel;
        MoveL E2,v100,z10,PM\WObj:=Pastel;
        MoveL E3,v100,z10,PM\WObj:=Pastel;
        MoveL E4,v100,z10,PM\WObj:=Pastel;
        MoveL E1,v100,z10,PM\WObj:=Pastel;
        MoveJ CUAA,v100,z10,PM\WObj:=Pastel;

    ENDPROC
    PROC Path_50()
        MoveJ P11,v50,z10,PM\WObj:=Pastel;
        MoveL P12,v50,z10,PM\WObj:=Pastel;
        MoveC P13,P14,v50,z10,PM\WObj:=Pastel;
        MoveC P15,P16,v50,z10,PM\WObj:=Pastel;
        MoveC P17,P18,v50,z10,PM\WObj:=Pastel;
        MoveC P19,P110,v50,z10,PM\WObj:=Pastel;
        MoveC P111,P112,v50,z10,PM\WObj:=Pastel;
        MoveC P113,P114,v50,z10,PM\WObj:=Pastel;
        MoveJ P115,v50,z10,PM\WObj:=Pastel;
        MoveL P116,v50,z10,PM\WObj:=Pastel;
        MoveL P117,v50,z10,PM\WObj:=Pastel;
        MoveC P118,P119,v50,z10,PM\WObj:=Pastel;
        MoveC P120,P12,v50,z10,PM\WObj:=Pastel;
        MoveJ P11,v50,z10,PM\WObj:=Pastel;
    ENDPROC
    PROC Path_60()

        MoveJ P21,v50,z10,PM\WObj:=Pastel;
        MoveL P22,v50,z10,PM\WObj:=Pastel;
        MoveL P23,v50,z10,PM\WObj:=Pastel;
        MoveC P24,P25,v50,z10,PM\WObj:=Pastel;
        MoveL P26,v50,z10,PM\WObj:=Pastel;
        MoveL P27,v50,z10,PM\WObj:=Pastel;
        MoveC P28,P29,v50,z10,PM\WObj:=Pastel;
        MoveC P210,P211,v50,z10,PM\WObj:=Pastel;
        MoveC P212,P213,v50,z10,PM\WObj:=Pastel;
        MoveC P214,P215,v50,z10,PM\WObj:=Pastel;
        MoveC P216,P217,v50,z10,PM\WObj:=Pastel;
        MoveC P218,P219,v50,z10,PM\WObj:=Pastel;
        MoveC P220,P221,v50,z10,PM\WObj:=Pastel;
        MoveC P222,P223,v50,z10,PM\WObj:=Pastel;
        MoveL P224,v50,z10,PM\WObj:=Pastel;
        MoveL P225,v50,z10,PM\WObj:=Pastel;
        MoveC P226,P227,v50,z10,PM\WObj:=Pastel;
        MoveC P228,P229,v50,z10,PM\WObj:=Pastel;
        MoveL P230,v50,z10,PM\WObj:=Pastel;
        MoveL P22,v50,z10,PM\WObj:=Pastel;
        MoveC P231,P232,v50,z10,PM\WObj:=Pastel;

    ENDPROC
    PROC Path_70()

        MoveJ P31,v50,z10,PM\WObj:=Pastel;
        MoveL P32,v50,z10,PM\WObj:=Pastel;
        MoveC P33,P34,v50,z10,PM\WObj:=Pastel;
        MoveL P35,v50,z10,PM\WObj:=Pastel;
        MoveC P36,P37,v50,z10,PM\WObj:=Pastel;
        MoveL P38,v50,z10,PM\WObj:=Pastel;
        MoveL P39,v50,z10,PM\WObj:=Pastel;
        MoveL P38,v50,z10,PM\WObj:=Pastel;
        MoveL P310,v50,z10,PM\WObj:=Pastel;
        MoveL P311,v50,z10,PM\WObj:=Pastel;
        MoveL P310,v50,z10,PM\WObj:=Pastel;
        MoveL P312,v50,z10,PM\WObj:=Pastel;
        MoveC P313,P314,v50,z10,PM\WObj:=Pastel;
        MoveL P315,v50,z10,PM\WObj:=Pastel;
        MoveJ P316,v50,z10,PM\WObj:=Pastel;
        MoveL P317,v50,z10,PM\WObj:=Pastel;
        MoveL P318,v50,z10,PM\WObj:=Pastel;
        MoveL P319,v50,z10,PM\WObj:=Pastel;
        MoveL P320,v50,z10,PM\WObj:=Pastel;
        MoveL P321,v50,z10,PM\WObj:=Pastel;
        MoveL P320,v50,z10,PM\WObj:=Pastel;
        MoveL P322,v50,z10,PM\WObj:=Pastel;
        MoveL P323,v50,z10,PM\WObj:=Pastel;
        MoveJ P324,v50,z10,PM\WObj:=Pastel;
        MoveJ P325,v50,z10,PM\WObj:=Pastel;
        MoveL P326,v50,z10,PM\WObj:=Pastel;
        MoveC P327,P328,v50,z10,PM\WObj:=Pastel;
        MoveC P329,P330,v50,z10,PM\WObj:=Pastel;
        MoveC P331,P328,v50,z10,PM\WObj:=Pastel;
        MoveC P331,P330,v50,z10,PM\WObj:=Pastel;
        MoveC P334,P333,v50,z10,PM\WObj:=Pastel;
        MoveJ P332,v50,z10,PM\WObj:=Pastel;


    ENDPROC
    PROC Path_80()

        MoveJ Target_10,v50,z10,PM\WObj:=Pastel;
        MoveL Target_20,v50,z10,PM\WObj:=Pastel;
        MoveC Target_30,Target_40,v50,z10,PM\WObj:=Pastel;
        MoveJ Target_50,v50,z10,PM\WObj:=Pastel;
        MoveJ Target_60,v50,z10,PM\WObj:=Pastel;
        MoveC Target_70,Target_80,v50,z10,PM\WObj:=Pastel;
        MoveJ Target_90,v50,z10,PM\WObj:=Pastel;
        MoveJ Target_100,v50,z10,PM\WObj:=Pastel;
        MoveC Target_110,Target_120,v50,z10,PM\WObj:=Pastel;
        MoveJ Target_130,v50,z10,PM\WObj:=Pastel;
        MoveJ Target_140,v50,z10,PM\WObj:=Pastel;
        MoveC Target_150,Target_160,v50,z10,PM\WObj:=Pastel;
        MoveJ Target_170,v50,z10,PM\WObj:=Pastel;
        MoveJ Target_180,v50,z10,PM\WObj:=Pastel;
        MoveC Target_190,Target_200,v50,z10,PM\WObj:=Pastel;
        MoveJ Target_210,v50,z10,PM\WObj:=Pastel;
        MoveJ Target_220,v50,z10,PM\WObj:=Pastel;
        MoveL Target_230,v50,z10,PM\WObj:=Pastel;
        MoveC Target_240,Target_250,v50,z10,PM\WObj:=Pastel;
        MoveL Target_220,v50,z10,PM\WObj:=Pastel;
        MoveJ Target_260,v50,z10,PM\WObj:=Pastel;
        MoveJ Target_270,v50,z10,PM\WObj:=Pastel;
        MoveC Target_280,Target_340,v50,z10,PM\WObj:=Pastel;
        MoveC Target_290,Target_270,v50,z10,PM\WObj:=Pastel;
        MoveJ Target_390,v50,z10,PM\WObj:=Pastel;
        MoveJ Target_370,v50,z10,PM\WObj:=Pastel;
        MoveL Target_350,v50,z10,PM\WObj:=Pastel;
        MoveC Target_310,Target_360,v50,z10,PM\WObj:=Pastel;
        MoveC Target_300,Target_350,v50,z10,PM\WObj:=Pastel;
        MoveJ Target_380,v50,z10,PM\WObj:=Pastel;
        MoveL Target_420,v50,z10,PM\WObj:=Pastel;
        MoveC Target_470,Target_480,v50,z10,PM\WObj:=Pastel;
        MoveC Target_490,Target_420,v50,z10,PM\WObj:=Pastel;
        MoveJ Target_400,v50,z10,PM\WObj:=Pastel;
        MoveL Target_410,v50,z10,PM\WObj:=Pastel;
        MoveC Target_440,Target_450,v50,z10,PM\WObj:=Pastel;
        MoveC Target_460,Target_410,v50,z10,PM\WObj:=Pastel;


    ENDPROC

    PROC Path_100()
        MoveL Target_500,v100,z10,PM\WObj:=Pastel;
    ENDPROC
ENDMODULE
